KUKA KRL program: sps.sub

&ACCESS RVO
&REL 102
&COMMENT PLC on control
DEF  SPS ( )
  ;FOLD DECLARATIONS
  ;FOLD BASISTECH DECL
  ;Automatik extern
  DECL STATE_T STAT
  DECL MODUS_T MODE
  ;ENDFOLD (BASISTECH DECL)
  ;FOLD USER DECL
  ; Please insert user defined declarations
  BOOL xFirstcycle

  ;ENDFOLD (USER DECL)
  ;ENDFOLD (DECLARATIONS)
  ;FOLD INI
  ;FOLD AUTOEXT INIT
  INTERRUPT DECL 91 WHEN $PRO_STATE1==#P_FREE DO RESET_OUT ()
  INTERRUPT ON 91
  $LOOP_MSG[]="                                                            "
  MODE=#SYNC
  $H_POS=$H_POS
  ;Automatik extern
  IF $MODE_OP==#EX THEN
    CWRITE($CMD,STAT,MODE,"RUN /R1/CELL()")
  ENDIF
  ;ENDFOLD (AUTOEXT INIT)
  ;FOLD BACKUPMANAGER PLC INIT
  BM_ENABLED = FALSE
  BM_OUTPUTVALUE = 0
  ;ENDFOLD (BACKUPMANAGER PLC INIT)
  ;FOLD USER INIT
  ; Please insert user defined initialization commands
    xFirstcycle = TRUE

  ;ENDFOLD (USER INIT)
  ;ENDFOLD (INI) = TRUE

  LOOP
    WAIT FOR NOT($POWER_FAIL)
    TORQUE_MONITORING()
    ;FOLD BACKUPMANAGER PLC
    IF BM_ENABLED THEN
      BM_OUTPUTSIGNAL = BM_OUTPUTVALUE
    ENDIF
    ;ENDFOLD (BACKUPMANAGER PLC)
;FOLD GRIPPERTECH PLC;%{E}%MKUKATPGRP,%CSPS,%VSPS,%P
  IF (ZANGEN_FUNKT>0) THEN
    H50 (5,AKT_ZANGE,DUMMY,GDEFAULT )
    ZANGEN_FUNKT=0
  ENDIF
;ENDFOLD (GRIPPERTECH PLC)

    ;FOLD USER PLC
    ; Subprogramms
    ; SPS_PROG(xFirstcycle, ..,..)

    ;ENDFOLD (USER PLC)

    xFirstcycle = FALSE
  ENDLOOP
  ;FOLD ;%{H}
  ;FOLD
END
  ;ENDFOLD


DEF  RESET_OUT ( )
  INT N
  MsgLoop(" ")
  IF REFLECT_PROG_NR == 1 THEN
    FOR N = 0 TO PGNO_LENGTH - 1
      $OUT[PGNO_FBIT_REFL + N] = FALSE
    ENDFOR
  ENDIF
  IF (PGNO_REQ>0) THEN
    $OUT[PGNO_REQ]=FALSE
  ELSE
    IF (PGNO_REQ<0) THEN
      $OUT[-PGNO_REQ]=TRUE
    ENDIF
  ENDIF
END

;FOLD USER SUBROUTINE
; Integrate your user defined subroutines

;ENDFOLD (USER SUBROUTINE)
;ENDFOLD
